DATA_BLOCK "dbArchiveParShipping"
{ S7_Optimized_Access := 'TRUE' }
VERSION : 0.8
NON_RETAIN
"fbArchiveParShipping"

BEGIN

END_DATA_BLOCK

